// TIA Portal V18 export
FUNCTION_BLOCK "auto_analog_copySpeed"   // FB22, FBD
{ S7_Optimized_Access := 'TRUE' }
VERSION : 0.1
// stored: AutoNumber true, IsIECCheckEnabled false, IsRetainMemResEnabled false, MemoryReserve 100, SetENOAutomatically false, UDAEnableTagReadback false
   VAR_INPUT
      ALLOWED : Bool;
      SET_SPD_wDir { ExternalAccessible := 'False'; ExternalVisible := 'False'; ExternalWritable := 'False'} : Real;
      MASTER_POS : Real;
      MY_POS : Real;
      par_max_Vcor : Real;
      par_max_Pos_delta : Real;
      xFwdOK : Bool;
      xRevOK : Bool;
      par_spd_absmax : Real;
      par_dist_absmax : Real;
      par_spd_crawl : Real;
      par_dist_crawl : Real;
      par_dist_stop : Real;
      par_lim_fwd : Real;
      par_lim_rev : Real;
      par_prec_au : Real;
      par_tout_follw : Time;
      par_SpeedTHreshold : Real;
      isMultiturn : Bool;
      MultiTurnGoesFwdOnly : Bool;
   END_VAR
   VAR_OUTPUT
      SPEED : Real;
      INPOS : Bool;
      ER_follow : Bool;
      ER_settings : Bool;
      ER_SET2 : Bool;
      ER_W : WString;
   END_VAR
   VAR
      should_move_static : Bool;
   END_VAR
   VAR_TEMP
      dir_fwd : Bool;
      dir_rev : Bool;
      arrived : Bool;
      distance : Real;
      estop_ok_no_err : Bool;
      speed_by_lag : Real;
      speed_by_lag_pos : Real;
      speed_out_abs : Real;
      xFWDREV_matter : Bool;
      limits_matter : Bool;
   END_VAR
BEGIN

REGION Network 2
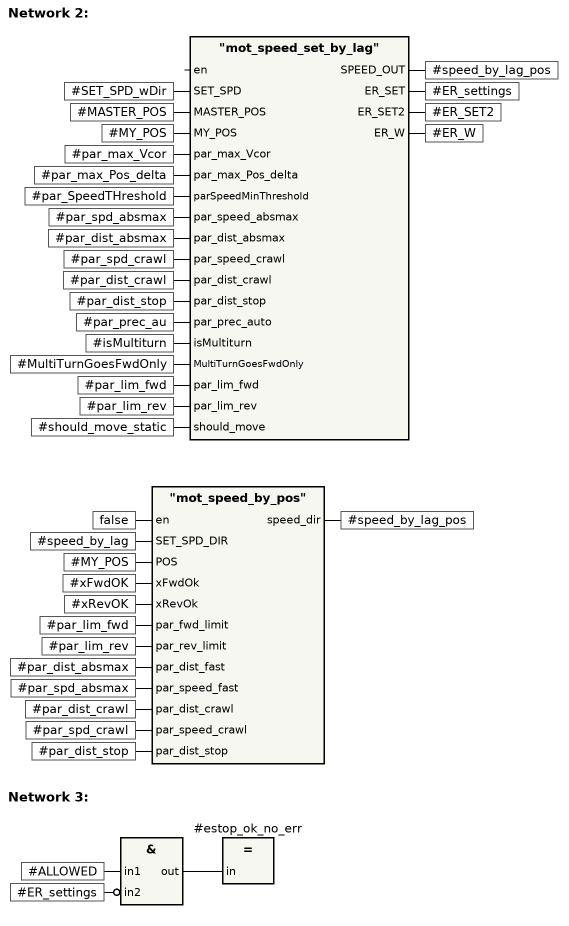
   "mot_speed_set_by_lag"(SET_SPD := #SET_SPD_wDir,
                          MASTER_POS := #MASTER_POS,
                          MY_POS := #MY_POS,
                          par_max_Vcor := #par_max_Vcor,
                          par_max_Pos_delta := #par_max_Pos_delta,
                          parSpeedMinThreshold := #par_SpeedTHreshold,
                          par_speed_absmax := #par_spd_absmax,
                          par_dist_absmax := #par_dist_absmax,
                          par_speed_crawl := #par_spd_crawl,
                          par_dist_crawl := #par_dist_crawl,
                          par_dist_stop := #par_dist_stop,
                          par_prec_auto := #par_prec_au,
                          isMultiturn := #isMultiturn,
                          MultiTurnGoesFwdOnly := #MultiTurnGoesFwdOnly,
                          par_lim_fwd := #par_lim_fwd,
                          par_lim_rev := #par_lim_rev,
                          should_move := #should_move_static,
                          SPEED_OUT => #speed_by_lag_pos,
                          ER_SET => #ER_settings,
                          ER_SET2 => #ER_SET2,
                          ER_W => #ER_W);
   IF false THEN
       "mot_speed_by_pos"(SET_SPD_DIR := #speed_by_lag,
                          POS := #MY_POS,
                          xFwdOk := #xFwdOK,
                          xRevOk := #xRevOK,
                          par_fwd_limit := #par_lim_fwd,
                          par_rev_limit := #par_lim_rev,
                          par_dist_fast := #par_dist_absmax,
                          par_speed_fast := #par_spd_absmax,
                          par_dist_crawl := #par_dist_crawl,
                          par_speed_crawl := #par_spd_crawl,
                          par_dist_stop := #par_dist_stop,
                          speed_dir => #speed_by_lag_pos);
   END_IF;
END_REGION

REGION Network 3
   #estop_ok_no_err := #ALLOWED AND NOT #ER_settings;
END_REGION

REGION Network 4 (SCL)
   #INPOS := ABS(#MASTER_POS - #MY_POS) < #par_prec_au;
END_REGION

REGION Network 5
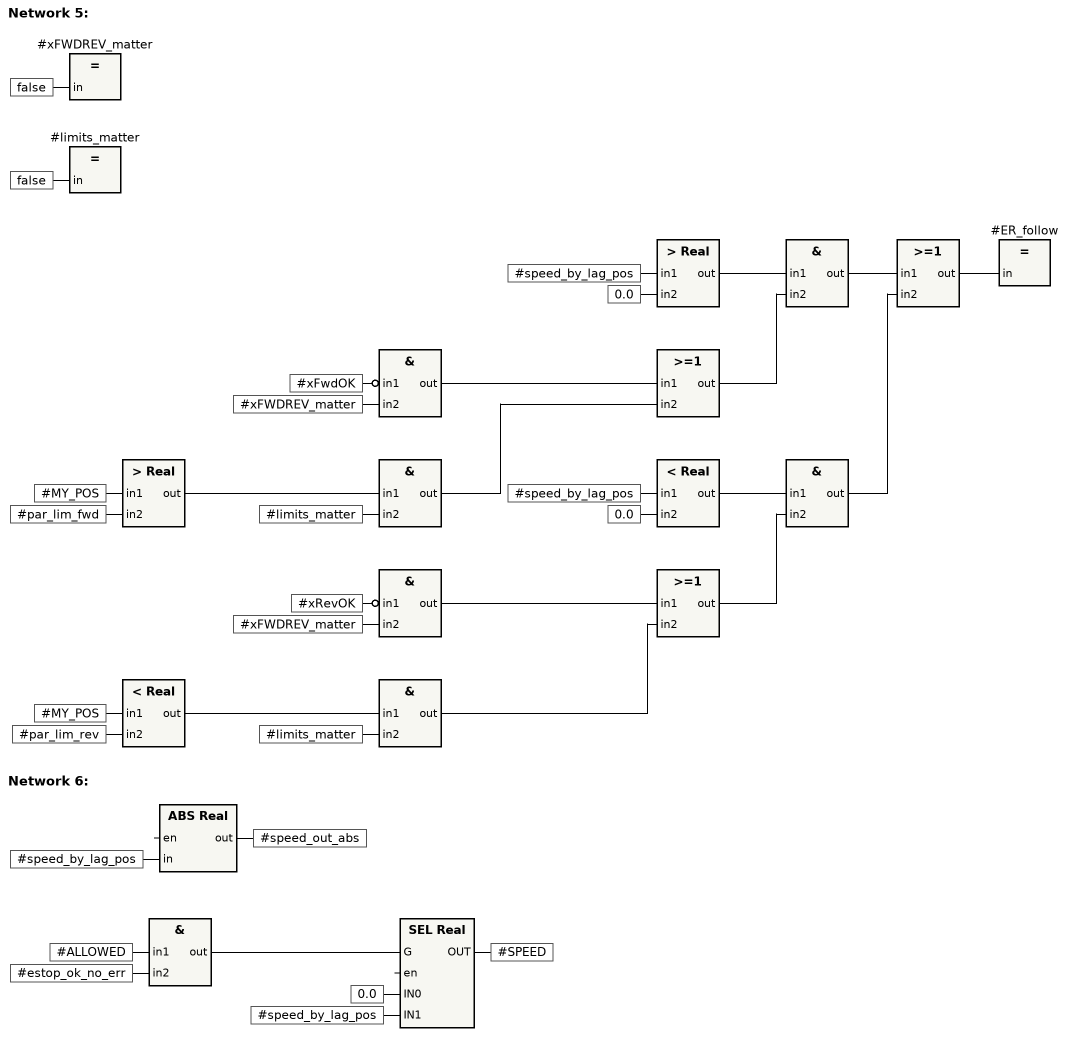
   #xFWDREV_matter := false;
   #limits_matter := false;
   #ER_follow := ((#speed_by_lag_pos > 0.0) AND ((NOT #xFwdOK AND #xFWDREV_matter) OR ((#MY_POS > #par_lim_fwd) AND #limits_matter))) OR ((#speed_by_lag_pos < 0.0) AND ((NOT #xRevOK AND #xFWDREV_matter) OR ((#MY_POS < #par_lim_rev) AND #limits_matter)));
END_REGION

REGION Network 6
   #speed_out_abs := ABS(#speed_by_lag_pos);
   #SPEED := SEL(G := #ALLOWED AND #estop_ok_no_err, IN0 := 0.0, IN1 := #speed_by_lag_pos);
END_REGION
END_FUNCTION_BLOCK
